(* CoDeSys 2.3 export: UDPOPENSENDSOCKET.EXP *)

(* POU Udp specific/UdpOpenSendSocket, ST *)
FUNCTION UdpOpenSendSocket : DINT
VAR_INPUT
	iPort:INT;
END_VAR
VAR
	diSocket:DINT;
	diOption:DINT;
END_VAR
(* @TEXT_IMPLEMENTATION := 'ST' *)
diSocket:=SysSockCreate(SOCKET_AF_INET, SOCKET_DGRAM, 0);
diOption:=1;
IF SysSockSetOption(diSocket, SOCKET_SOL, SOCKET_SO_BROADCAST, ADR(diOption), SIZEOF(diOption)) = FALSE THEN
	UdpOpenSendSocket:=SOCKET_INVALID;
ELSE
	UdpOpenSendSocket:=diSocket;
END_IF
END_FUNCTION
